{attribute addProperty BoxType "EL2262-0000-0002"}
{attribute addProperty Id "Cycle_Counter1AT %Q*UINT162"}
{attribute addProperty CRC "2005400093"}
{attribute addProperty SizeInBites "16"}
{attribute addProperty SizeInBytes "2"}
TYPE CycCount1_7787FA1D :
STRUCT
	{attribute addProperty Name "Cycle_Counter1"}
	Cycle_Counter1 AT %Q* : UINT;
END_STRUCT
END_TYPE

(* stored: Version 1.2.0.0, ProductVersion 3.1.4024.9
   DUT CycCount1_7787FA1D: Id {ac81e8e3-0432-42ac-8b13-a61858c494ed} *)
